FUNCTION_BLOCK MasterMove
VAR_INPUT
	MoveDistance		: LREAL;
	MoveVelocity			: LREAL;
	MoveAcceleration		: LREAL;
	MoveDeceleration		: LREAL;
	MoveJerk			: LREAL;
END_VAR
VAR_OUTPUT
END_VAR
VAR
END_VAR


Master.fbMC_MoveRelative[1](
	Execute  		:= TRUE,
	Distance		:= MoveDistance,
	Velocity  		:= MoveVelocity,
	Acceleration   := MoveAcceleration,
	Deceleration  := MoveDeceleration,
	Jerk			:= MoveJerk,
	BufferMode     := MC_BlendingHigh,
	Axis			:= Master.Axis
);

Master.fbMC_MoveRelative[1](
	Execute  		:= FALSE,
	Axis			:= Master.Axis
);

END_FUNCTION_BLOCK

(* stored: Version 1.1.0.1, ProductVersion 3.1.4024.9
   POU MasterMove: Id {d890bfe9-b53a-44dd-929c-9bbbef9d41f0}, SpecialFunc None *)
